FUNCTION_BLOCK FB_HeartbeatMonitor
VAR_INPUT
	CLK	: BOOL;
	PT	: TIME := T#2S;
END_VAR
VAR_OUTPUT
	Q	: BOOL;
END_VAR
VAR
	fbHbTimeout: TON;
	bLastHB: BOOL;
	bFirstBeatRec	: BOOL;
END_VAR

IF bLastHB <> CLK THEN
	bFirstBeatRec := TRUE;
END_IF

fbHbTimeout(IN:= (bLastHB = CLK), PT:= PT, Q=> Q, ET=> );
Q := NOT fbHbTimeout.Q AND bFirstBeatRec;
bLastHB := CLK;

END_FUNCTION_BLOCK

(* stored: Version 1.1.0.1, ProductVersion 3.1.4024.9
   POU FB_HeartbeatMonitor: Id {e8b36ecf-1680-4703-ae1e-ebe9f8b4fe16}, SpecialFunc None *)
